FUNCTION Norm_x_UINT : REAL
VAR_INPUT
	raw_input : REAL;
	x_max : UINT := 32767;  //for AI, use 32767, for AQ, use 12,000 or 50,000 V.
	x_min : UINT := 0;
END_VAR
VAR
END_VAR

// 0 - 12kV or 50kV input 
Norm_x_UINT := (raw_input - x_min) / (x_max - x_min);

END_FUNCTION

(* stored: Version 1.1.0.1, ProductVersion 3.1.4024.9
   POU Norm_x_UINT: Id {5fc247a3-a867-4ccf-9b47-196535dbc4e0}, SpecialFunc None *)
